FUNCTION_BLOCK RegisterService (* Register Service Function Block *)
  (* Standard: 61499-2; Description: Copyright (c) 2018 fortiss GmbH This program and the accompanying materials are made available under the terms of the Eclipse Public License 2.0 which is available at https://www.eclipse.org/legal/epl-2.0/ SPDX-License-Identifier: EPL-2.0 *)
  (* Version 1.0, 2018-09-21, Jose Cabral, fortiss GmbH *)
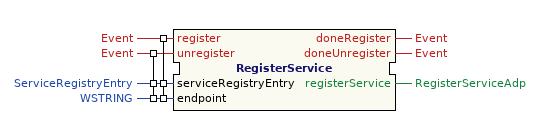
  EVENT_INPUT
    register WITH serviceRegistryEntry, endpoint; (* Register the service *)
    unregister WITH serviceRegistryEntry, endpoint; (* Unregister the service *)
  END_EVENT
  EVENT_OUTPUT
    doneRegister; (* Register finished *)
    doneUnregister; (* Unregister finished *)
  END_EVENT
  VAR_INPUT
    serviceRegistryEntry : ServiceRegistryEntry; (* Service Registry Entry for register or unregister *)
    endpoint : WSTRING; (* Endpoint (IP:PORT/URI) of the Service Registry (not officially in the documentation, but it simplifies the FBs) *)
  END_VAR
  PLUGS
    registerService : RegisterServiceAdp; (* Register service adapter *)
  END_PLUGS
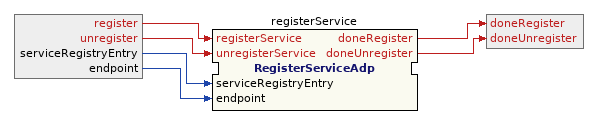
  EVENT_CONNECTIONS
    register TO registerService.registerService;
    unregister TO registerService.unregisterService;
    registerService.doneRegister TO doneRegister;
    registerService.doneUnregister TO doneUnregister;
  END_CONNECTIONS
  DATA_CONNECTIONS
    serviceRegistryEntry TO registerService.serviceRegistryEntry;
    endpoint TO registerService.endpoint;
  END_CONNECTIONS
END_FUNCTION_BLOCK
